KUKA KRL program: ho_st600_r1_1_2.src, ho_st600_r1_1_2.dat

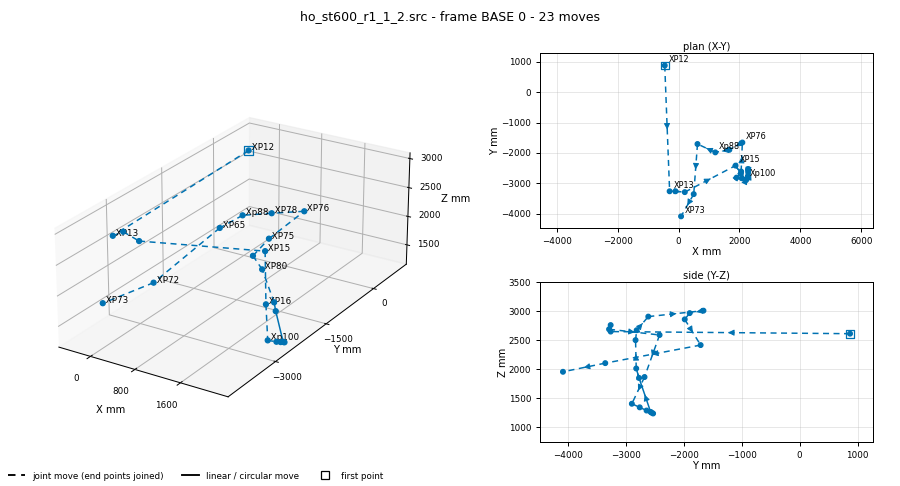
[picture p0: tool path of ho_st600_r1_1_2.src in frame BASE 0, 23 of 23 moves have a stored position in this frame; points joined in program order, loops and branches not executed]
--- ho_st600_r1_1_2.src ---
&ACCESS RVO1
&REL 137
&COMMENT Pega traseira ACTROS
&PARAM DISKPATH = KRC:\R1\Program\MANIPULACAO LTC
DEF ho_st600_r1_1_2( )
;FOLD INI
  ;FOLD BASISTECH INI
    GLOBAL INTERRUPT DECL 3 WHEN $STOPMESS==TRUE DO IR_STOPM ( )
    INTERRUPT ON 3
    BAS (#INITMOV,0 )
  ;ENDFOLD (BASISTECH INI)
;FOLD GRIPPERTECH INI
USER_GRP(0,DUMMY,DUMMY,GDEFAULT)
;ENDFOLD (GRIPPERTECH INI)
  ;FOLD USER INI
    ;Make your modifications here

  ;ENDFOLD (USER INI)
;ENDFOLD (INI)

; Caracterização dos meios de produção:
; Changes: Pega Traseira Actros
; Modelos: MGS\MGSB\LTA\LTB\STB
; Versão Atual: 22/07/2015
; Name: P13.050-R1

chk_w5_wechs_ok ( )              ; CHECK GRIPPER ACTROS

;FOLD PTP P12 CONT Vel=100 % PDAT11 Tool[5]:Painel Traseiro Actros Base[0];%{PE}%R 8.2.19,%MKUKATPBASIS,%CMOVE,%VPTP,%P 1:PTP, 2:P12, 3:C_DIS, 5:100, 7:PDAT11
$BWDSTART=FALSE
PDAT_ACT=PPDAT11
FDAT_ACT=FP12
BAS(#PTP_PARAMS,100)
PTP XP12 C_DIS
;ENDFOLD
;FOLD PTP P13 Vel=100 % PDAT12 Tool[5]:Painel Traseiro Actros Base[0];%{PE}%R 8.2.20,%MKUKATPBASIS,%CMOVE,%VPTP,%P 1:PTP, 2:P13, 3:, 5:100, 7:PDAT12
$BWDSTART=FALSE
PDAT_ACT=PPDAT12
FDAT_ACT=FP13
BAS(#PTP_PARAMS,100)
PTP XP13
;ENDFOLD

;FOLD OUT 3352 'R1 busca traseira' State=TRUE ;%{PE}%R 8.2.20,%MKUKATPBASIS,%COUT,%VOUTX,%P 2:3352, 3:R1 busca traseira, 5:TRUE, 6:
$OUT[3352]=TRUE
;ENDFOLD
;FOLD WAIT FOR ( IN 3352 'Aguarda lib. Buscar traseira' );%{PE}%R 8.2.20,%MKUKATPBASIS,%CEXT_WAIT_FOR,%VEXT_WAIT_FOR,%P 2:, 4:, 5:$IN, 6:3352, 7:Aguarda lib. Buscar traseira, 9:
WAIT FOR  ( $IN[3352] )
;ENDFOLD
;FOLD OUT 3352 'R1 busca traseira' State=FALSE ;%{PE}%R 8.2.20,%MKUKATPBASIS,%COUT,%VOUTX,%P 2:3352, 3:R1 busca traseira, 5:FALSE, 6:
$OUT[3352]=FALSE
;ENDFOLD

;FOLD PTP P74 Vel=100 % PDAT78 Tool[5]:Painel Traseiro Actros Base[0];%{PE}%R 8.2.20,%MKUKATPBASIS,%CMOVE,%VPTP,%P 1:PTP, 2:P74, 3:, 5:100, 7:PDAT78
$BWDSTART=FALSE
PDAT_ACT=PPDAT78
FDAT_ACT=FP74
BAS(#PTP_PARAMS,100)
PTP XP74
;ENDFOLD
;FOLD PTP P14 CONT Vel=100 % PDAT13 Tool[5]:Painel Traseiro Actros Base[0];%{PE}%R 8.2.19,%MKUKATPBASIS,%CMOVE,%VPTP,%P 1:PTP, 2:P14, 3:C_DIS, 5:100, 7:PDAT13
$BWDSTART=FALSE
PDAT_ACT=PPDAT13
FDAT_ACT=FP14
BAS(#PTP_PARAMS,100)
PTP XP14 C_DIS
;ENDFOLD
;FOLD PTP P15 CONT Vel=100 % PDAT14 Tool[5]:Painel Traseiro Actros Base[0];%{PE}%R 8.2.19,%MKUKATPBASIS,%CMOVE,%VPTP,%P 1:PTP, 2:P15, 3:C_DIS, 5:100, 7:PDAT14
$BWDSTART=FALSE
PDAT_ACT=PPDAT14
FDAT_ACT=FP15
BAS(#PTP_PARAMS,100)
PTP XP15 C_DIS
;ENDFOLD
;FOLD PTP P16 CONT Vel=100 % PDAT15 Tool[5]:Painel Traseiro Actros Base[0];%{PE}%R 8.2.19,%MKUKATPBASIS,%CMOVE,%VPTP,%P 1:PTP, 2:P16, 3:C_DIS, 5:100, 7:PDAT15
$BWDSTART=FALSE
PDAT_ACT=PPDAT15
FDAT_ACT=FP16
BAS(#PTP_PARAMS,100)
PTP XP16 C_DIS
;ENDFOLD

;FOLD OUT 3342 'Fora area externa' State=FALSE ;%{PE}%R 8.2.20,%MKUKATPBASIS,%COUT,%VOUTX,%P 2:3342, 3:Fora area externa, 5:FALSE, 6:
$OUT[3342]=FALSE
;ENDFOLD

;FOLD SET Z2.1/2 GRP ACTROS State= GDAT2;%{PE}%R 8.2.1,%MKUKATPGRP,%CGRP,%VGRP,%P 2:1, 4:1, 5:#NO, 6:GDAT2, 8:0, 10:0
H50(GRP,1,1,GGDAT2)
;ENDFOLD
chk_w5_grp2_opn()
;FOLD SET Z3.1/2 GRP ACTROS State=OPN GDAT3;%{PE}%R 8.2.1,%MKUKATPGRP,%CGRP,%VGRP,%P 2:2, 4:1, 5:#NO, 6:GDAT3, 8:0, 10:0
H50(GRP,2,1,GGDAT3)
;ENDFOLD
chk_w5_grp3_opn()

;FOLD PTP p100 CONT Vel=100 % PDAT71 Tool[5]:Painel Traseiro Actros Base[0];%{PE}%R 8.2.20,%MKUKATPBASIS,%CMOVE,%VPTP,%P 1:PTP, 2:p100, 3:C_DIS, 5:100, 7:PDAT71
$BWDSTART=FALSE
PDAT_ACT=PPDAT71
FDAT_ACT=Fp100
BAS(#PTP_PARAMS,100)
PTP Xp100 C_DIS
;ENDFOLD
;FOLD PTP p102 CONT Vel=100 % PDAT73 Tool[5]:Painel Traseiro Actros Base[0];%{PE}%R 8.2.20,%MKUKATPBASIS,%CMOVE,%VPTP,%P 1:PTP, 2:p102, 3:C_DIS, 5:100, 7:PDAT73
$BWDSTART=FALSE
PDAT_ACT=PPDAT73
FDAT_ACT=Fp102
BAS(#PTP_PARAMS,100)
PTP Xp102 C_DIS
;ENDFOLD
;FOLD PTP P82 Vel=100 % PDAT84 Tool[5]:Painel Traseiro Actros Base[0];%{PE}%R 8.2.20,%MKUKATPBASIS,%CMOVE,%VPTP,%P 1:PTP, 2:P82, 3:, 5:100, 7:PDAT84
$BWDSTART=FALSE
PDAT_ACT=PPDAT84
FDAT_ACT=FP82
BAS(#PTP_PARAMS,100)
PTP XP82
;ENDFOLD

;FOLD ; POSICAO DE PEGA DA PECA;%{PE}%R 8.2.20,%MKUKATPBASIS,%CCOMMENT,%VNORMAL,%P 2:POSICAO  DE  PEGA  DA  PECA
;ENDFOLD
;FOLD LIN P18 Vel=0.5 m/s CPDAT1 Tool[5]:Painel Traseiro Actros Base[0];%{PE}%R 8.2.20,%MKUKATPBASIS,%CMOVE,%VLIN,%P 1:LIN, 2:P18, 3:, 5:0.5, 7:CPDAT1
$BWDSTART=FALSE
LDAT_ACT=LCPDAT1
FDAT_ACT=FP18
BAS(#CP_PARAMS,0.5)
LIN XP18
;ENDFOLD

IF (NOT(GHOST())) THEN
;FOLD WAIT FOR ( IN 1 'Presença de peça 1 - Actros Todos' ) AND ( IN 2 'Presença de peça 2 - Actros Todos' );%{PE}%R 8.2.20,%MKUKATPBASIS,%CEXT_WAIT_FOR,%VEXT_WAIT_FOR,%P 2:, 4:, 5:$IN, 6:1, 7:Presença de peça 1 - Actros Todos, 9:AND, 10:, 12:, 13:$IN, 14:2, 15:Presença de peça 2 - Actros Todos, 17:
WAIT FOR  ( $IN[1] ) AND ( $IN[2] )
;ENDFOLD
ENDIF

;FOLD SET Z2.1/2 GRP ACTROS State=CLO GDAT1;%{PE}%R 8.2.1,%MKUKATPGRP,%CGRP,%VGRP,%P 2:1, 4:2, 5:#NO, 6:GDAT1, 8:0, 10:0
H50(GRP,1,2,GGDAT1)
;ENDFOLD
chk_w5_grp2_clo()
;FOLD SET Z3.1/2 GRP ACTROS State=CLO GDAT4;%{PE}%R 8.2.1,%MKUKATPGRP,%CGRP,%VGRP,%P 2:2, 4:2, 5:#NO, 6:GDAT4, 8:0, 10:0
H50(GRP,2,2,GGDAT4)
;ENDFOLD
chk_w5_grp3_clo()

IF (NOT(GHOST())) THEN
;FOLD SET Ventosa ACTROS State=VACUUM GDAT5;%{PE}%R 8.2.1,%MKUKATPGRP,%CGRP,%VGRP,%P 2:6, 4:1, 5:#NO, 6:GDAT5, 8:0, 10:0
H50(GRP,6,1,GGDAT5)
;ENDFOLD
;chk_w5_grp1_vac()
ENDIF

;FOLD OUT 3349 'R1 pegou peça' State=TRUE ;%{PE}%R 8.2.20,%MKUKATPBASIS,%COUT,%VOUTX,%P 2:3349, 3:R1 pegou peça, 5:TRUE, 6:
$OUT[3349]=TRUE
;ENDFOLD
;FOLD OUT 3350 'Solicita lib. sair magazine' State=TRUE ;%{PE}%R 8.2.20,%MKUKATPBASIS,%COUT,%VOUTX,%P 2:3350, 3:Solicita lib. sair magazine, 5:TRUE, 6:
$OUT[3350]=TRUE
;ENDFOLD
;FOLD WAIT FOR ( IN 3349 'Aguarda lib sair magazine' );%{PE}%R 8.2.20,%MKUKATPBASIS,%CEXT_WAIT_FOR,%VEXT_WAIT_FOR,%P 2:, 4:, 5:$IN, 6:3349, 7:Aguarda lib sair magazine, 9:
WAIT FOR  ( $IN[3349] )
;ENDFOLD
;FOLD OUT 3350 'Solicita lib sair magazine' State=FALSE ;%{PE}%R 8.2.20,%MKUKATPBASIS,%COUT,%VOUTX,%P 2:3350, 3:Solicita lib sair magazine, 5:FALSE, 6:
$OUT[3350]=FALSE
;ENDFOLD

;FOLD LIN P81 CONT Vel=1 m/s CPDAT16 Tool[5]:Painel Traseiro Actros Base[0];%{PE}%R 8.2.20,%MKUKATPBASIS,%CMOVE,%VLIN,%P 1:LIN, 2:P81, 3:C_DIS C_DIS, 5:1, 7:CPDAT16
$BWDSTART=FALSE
LDAT_ACT=LCPDAT16
FDAT_ACT=FP81
BAS(#CP_PARAMS,1)
LIN XP81 C_DIS C_DIS
;ENDFOLD
;FOLD LIN p101 CONT Vel=1 m/s CPDAT12 Tool[5]:Painel Traseiro Actros Base[0];%{PE}%R 8.2.20,%MKUKATPBASIS,%CMOVE,%VLIN,%P 1:LIN, 2:p101, 3:C_DIS C_DIS, 5:1, 7:CPDAT12
$BWDSTART=FALSE
LDAT_ACT=LCPDAT12
FDAT_ACT=Fp101
BAS(#CP_PARAMS,1)
LIN Xp101 C_DIS C_DIS
;ENDFOLD
;FOLD LIN P79 CONT Vel=2 m/s CPDAT15 Tool[5]:Painel Traseiro Actros Base[0];%{PE}%R 8.2.20,%MKUKATPBASIS,%CMOVE,%VLIN,%P 1:LIN, 2:P79, 3:C_DIS C_DIS, 5:2, 7:CPDAT15
$BWDSTART=FALSE
LDAT_ACT=LCPDAT15
FDAT_ACT=FP79
BAS(#CP_PARAMS,2)
LIN XP79 C_DIS C_DIS
;ENDFOLD
;FOLD LIN p95 CONT Vel=1 m/s CPDAT11 Tool[5]:Painel Traseiro Actros Base[0];%{PE}%R 8.2.20,%MKUKATPBASIS,%CMOVE,%VLIN,%P 1:LIN, 2:p95, 3:C_DIS C_DIS, 5:1, 7:CPDAT11
$BWDSTART=FALSE
LDAT_ACT=LCPDAT11
FDAT_ACT=Fp95
BAS(#CP_PARAMS,1)
LIN Xp95 C_DIS C_DIS
;ENDFOLD

IF (NOT(GHOST())) THEN
;FOLD WAIT FOR ( IN 1 'Presença de peça 1 - Actros Todos' ) AND ( IN 2 'Presença de peça 2 - Actros Todos' );%{PE}%R 8.2.20,%MKUKATPBASIS,%CEXT_WAIT_FOR,%VEXT_WAIT_FOR,%P 2:, 4:, 5:$IN, 6:1, 7:Presença de peça 1 - Actros Todos, 9:AND, 10:, 12:, 13:$IN, 14:2, 15:Presença de peça 2 - Actros Todos, 17:
WAIT FOR  ( $IN[1] ) AND ( $IN[2] )
;ENDFOLD
ENDIF

;FOLD PTP P80 CONT Vel=100 % PDAT83 Tool[5]:Painel Traseiro Actros Base[0];%{PE}%R 8.2.20,%MKUKATPBASIS,%CMOVE,%VPTP,%P 1:PTP, 2:P80, 3:C_DIS, 5:100, 7:PDAT83
$BWDSTART=FALSE
PDAT_ACT=PPDAT83
FDAT_ACT=FP80
BAS(#PTP_PARAMS,100)
PTP XP80 C_DIS
;ENDFOLD
;FOLD PTP P21 CONT Vel=100 % PDAT19 Tool[5]:Painel Traseiro Actros Base[0];%{PE}%R 8.2.19,%MKUKATPBASIS,%CMOVE,%VPTP,%P 1:PTP, 2:P21, 3:C_DIS, 5:100, 7:PDAT19
$BWDSTART=FALSE
PDAT_ACT=PPDAT19
FDAT_ACT=FP21
BAS(#PTP_PARAMS,100)
PTP XP21 C_DIS
;ENDFOLD
;FOLD PTP P75 CONT Vel=100 % PDAT79 Tool[5]:Painel Traseiro Actros Base[0];%{PE}%R 8.2.20,%MKUKATPBASIS,%CMOVE,%VPTP,%P 1:PTP, 2:P75, 3:C_DIS, 5:100, 7:PDAT79
$BWDSTART=FALSE
PDAT_ACT=PPDAT79
FDAT_ACT=FP75
BAS(#PTP_PARAMS,100)
PTP XP75 C_DIS
;ENDFOLD
;FOLD PTP P76 CONT Vel=100 % PDAT80 Tool[5]:Painel Traseiro Actros Base[0];%{PE}%R 8.2.20,%MKUKATPBASIS,%CMOVE,%VPTP,%P 1:PTP, 2:P76, 3:C_DIS, 5:100, 7:PDAT80
$BWDSTART=FALSE
PDAT_ACT=PPDAT80
FDAT_ACT=FP76
BAS(#PTP_PARAMS,100)
PTP XP76 C_DIS
;ENDFOLD
;FOLD PTP P78 CONT Vel=100 % PDAT82 Tool[5]:Painel Traseiro Actros Base[0];%{PE}%R 8.2.20,%MKUKATPBASIS,%CMOVE,%VPTP,%P 1:PTP, 2:P78, 3:C_DIS, 5:100, 7:PDAT82
$BWDSTART=FALSE
PDAT_ACT=PPDAT82
FDAT_ACT=FP78
BAS(#PTP_PARAMS,100)
PTP XP78 C_DIS
;ENDFOLD
;FOLD PTP p88 CONT Vel=100 % PDAT60 Tool[5]:Painel Traseiro Actros Base[0];%{PE}%R 8.2.19,%MKUKATPBASIS,%CMOVE,%VPTP,%P 1:PTP, 2:p88, 3:C_DIS, 5:100, 7:PDAT60
$BWDSTART=FALSE
PDAT_ACT=PPDAT60
FDAT_ACT=Fp88
BAS(#PTP_PARAMS,100)
PTP Xp88 C_DIS
;ENDFOLD
;FOLD PTP P65 CONT Vel=100 % PDAT74 Tool[5]:Painel Traseiro Actros Base[0];%{PE}%R 8.2.20,%MKUKATPBASIS,%CMOVE,%VPTP,%P 1:PTP, 2:P65, 3:C_DIS, 5:100, 7:PDAT74
$BWDSTART=FALSE
PDAT_ACT=PPDAT74
FDAT_ACT=FP65
BAS(#PTP_PARAMS,100)
PTP XP65 C_DIS
;ENDFOLD
;FOLD PTP P72 CONT Vel=100 % PDAT76 Tool[5]:Painel Traseiro Actros Base[0];%{PE}%R 8.2.20,%MKUKATPBASIS,%CMOVE,%VPTP,%P 1:PTP, 2:P72, 3:C_DIS, 5:100, 7:PDAT76
$BWDSTART=FALSE
PDAT_ACT=PPDAT76
FDAT_ACT=FP72
BAS(#PTP_PARAMS,100)
PTP XP72 C_DIS
;ENDFOLD

;FOLD Collision.Monitoring_AREA_5_On ;%{PE}%MKUKATPUSER
COLLSTOP( 11, 1 ) ;not Interrupt-Controlled
;ENDFOLD

;FOLD OUT 3349 'R1 Pegou peca' State=TRUE ;%{PE}%R 8.2.20,%MKUKATPBASIS,%COUT,%VOUTX,%P 2:3349, 3:R1 Pegou peca, 5:TRUE, 6:
$OUT[3349]=TRUE
;ENDFOLD
;FOLD OUT 3342 'Fora area externa' State=TRUE ;%{PE}%R 8.2.20,%MKUKATPBASIS,%COUT,%VOUTX,%P 2:3342, 3:Fora area externa, 5:TRUE, 6:
$OUT[3342]=TRUE
;ENDFOLD

;FOLD PTP P73 Vel=100 % PDAT77 Tool[5]:Painel Traseiro Actros Base[0];%{PE}%R 8.2.20,%MKUKATPBASIS,%CMOVE,%VPTP,%P 1:PTP, 2:P73, 3:, 5:100, 7:PDAT77
$BWDSTART=FALSE
PDAT_ACT=PPDAT77
FDAT_ACT=FP73
BAS(#PTP_PARAMS,100)
PTP XP73
;ENDFOLD

END

--- ho_st600_r1_1_2.dat ---
&ACCESS RVO1
&REL 137
&COMMENT Pega traseira ACTROS
&PARAM DISKPATH = KRC:\R1\Program\MANIPULACAO LTC
DEFDAT  ho_st600_r1_1_2
;FOLD EXTERNAL DECLARATIONS;%{PE}%MKUKATPBASIS,%CEXT,%VCOMMON,%P
;FOLD GRIPPERTECH EXT
EXT  H50 (INT  :IN,INT  :IN,INT  :IN,GRP_TYP  :IN )
;ENDFOLD (GRIPPERTECH EXT)
;FOLD SPOTTECH EXT
EXT  USERSPOT (S_COMMAND  :IN,SPOT_TYPE  :IN )
;ENDFOLD (SPOTTECH EXT)
;FOLD BASISTECH EXT;%{PE}%MKUKATPBASIS,%CEXT,%VEXT,%P
EXT  BAS (BAS_COMMAND  :IN,REAL  :IN )
DECL INT SUCCESS
;ENDFOLD (BASISTECH EXT)
;FOLD USER EXT;%{E}%MKUKATPUSER,%CEXT,%VEXT,%P
;Make your modifications here

;ENDFOLD (USER EXT)
;ENDFOLD (EXTERNAL DECLARATIONS)

;# ============ START PATH : bh_p13050r1_lta_01 =============
DECL BASIS_SUGG_T LAST_BASIS={POINT1[] "P82                     ",POINT2[] "P82                     ",CP_PARAMS[] "CPDAT0                  ",PTP_PARAMS[] "PDAT84                  ",CONT[] "                        ",CP_VEL[] "2.0                     ",PTP_VEL[] "100                     ",SYNC_PARAMS[] "SYNCDAT                 ",SPL_NAME[] "S0                      "}
DECL PDAT PPDAT11={VEL 100.0,ACC 100.0,APO_DIST 100.0,APO_MODE #CDIS}
DECL E6POS XP12={X -451.816589,Y 870.27887,Z 2616.43896,A -71.9595718,B 86.8192902,C 144.022598,S 2,T 11,E1 -267.097687,E2 0.0,E3 0.0,E4 0.0,E5 0.0,E6 0.0}
DECL FDAT FP12={TOOL_NO 5,BASE_NO 0,IPO_FRAME #BASE,POINT2[] " ",TQ_STATE FALSE}
DECL PDAT PPDAT12={VEL 100.0,ACC 100.0,APO_DIST 100.0,APO_MODE #CDIS}
DECL E6POS XP13={X -291.739288,Y -3257.74512,Z 2653.0061,A 20.6638298,B 86.1274414,C -123.413696,S 2,T 11,E1 -4438.05518,E2 0.0,E3 0.0,E4 0.0,E5 0.0,E6 0.0}
DECL FDAT FP13={TOOL_NO 5,BASE_NO 0,IPO_FRAME #BASE,POINT2[] " ",TQ_STATE FALSE}
DECL PDAT PPDAT13={VEL 100.0,ACC 100.0,APO_DIST 100.0,APO_MODE #CDIS}
DECL E6POS XP14={X 205.846802,Y -3285.1731,Z 2693.19409,A -3.17952704,B 85.6848679,C -123.935898,S 2,T 11,E1 -4438.06104,E2 0.0,E3 0.0,E4 0.0,E5 0.0,E6 0.0}
DECL FDAT FP14={TOOL_NO 5,BASE_NO 0,IPO_FRAME #BASE,POINT2[] " ",TQ_STATE FALSE}
DECL PDAT PPDAT14={VEL 100.0,ACC 100.0,APO_DIST 100.0,APO_MODE #CDIS}
DECL E6POS XP15={X 1872.49097,Y -2414.4231,Z 2594.0769,A -19.4102993,B 84.5822067,C -109.933098,S 2,T 11,E1 -3412.81689,E2 0.0,E3 0.0,E4 0.0,E5 0.0,E6 0.0}
DECL FDAT FP15={TOOL_NO 5,BASE_NO 0,IPO_FRAME #BASE,POINT2[] " ",TQ_STATE FALSE}
DECL PDAT PPDAT15={VEL 100.0,ACC 100.0,APO_DIST 100.0,APO_MODE #CDIS}
DECL E6POS XP16={X 2049.04297,Y -2673.92407,Z 1868.73901,A -84.6288071,B 74.7002335,C -174.507401,S 2,T 11,E1 -3291.271,E2 0.0,E3 0.0,E4 0.0,E5 0.0,E6 0.0}
DECL FDAT FP16={TOOL_NO 5,BASE_NO 0,IPO_FRAME #BASE,POINT2[] " ",TQ_STATE FALSE}
DECL LDAT LCPDAT1={VEL 2.0,ACC 100.0,APO_DIST 100.0,APO_FAC 50.0,AXIS_VEL 100.0,AXIS_ACC 100.0,ORI_TYP #VAR,CIRC_TYP #BASE,JERK_FAC 50.0,GEAR_JERK 50.0,EXAX_IGN 0}
DECL E6POS XP18={X 2287.61304,Y -2526.11206,Z 1240.37695,A -89.8074493,B 66.0794296,C -179.626907,S 2,T 11,E1 -3241.46289,E2 0.0,E3 0.0,E4 0.0,E5 0.0,E6 0.0}
DECL FDAT FP18={TOOL_NO 5,BASE_NO 0,IPO_FRAME #BASE,POINT2[] " ",TQ_STATE FALSE}
DECL E6POS XP21={X 1903.797,Y -2809.604,Z 2675.91406,A -52.9545403,B 81.9597015,C -137.800507,S 2,T 11,E1 -3600.21191,E2 0.0,E3 0.0,E4 0.0,E5 0.0,E6 0.0}
DECL FDAT FP21={TOOL_NO 5,BASE_NO 0,IPO_FRAME #BASE,POINT2[] " ",TQ_STATE FALSE}
DECL PDAT PPDAT19={VEL 100.0,ACC 100.0,APO_DIST 100.0,APO_MODE #CDIS}
DECL E6POS XP88={X 1207.65796,Y -1980.32104,Z 2863.53809,A 30.6810093,B 83.3284302,C 30.6459599,S 2,T 10,E1 -964.773499,E2 0.0,E3 0.0,E4 0.0,E5 0.0,E6 0.0}
DECL FDAT Fp88={TOOL_NO 5,BASE_NO 0,IPO_FRAME #BASE,POINT2[] " ",TQ_STATE FALSE}
DECL PDAT PPDAT60={VEL 100.0,ACC 100.0,APO_DIST 100.0,APO_MODE #CDIS}
DECL E6POS XP95={X 2276.68311,Y -2816.91406,Z 2016.46301,A -88.0621414,B 73.5641479,C -177.631104,S 2,T 11,E1 -3601.14893,E2 0.0,E3 0.0,E4 0.0,E5 0.0,E6 0.0}
DECL FDAT Fp95={TOOL_NO 5,BASE_NO 0,IPO_FRAME #BASE,POINT2[] " ",TQ_STATE FALSE}
DECL LDAT LCPDAT11={VEL 2.0,ACC 100.0,APO_DIST 100.0,APO_FAC 50.0,AXIS_VEL 100.0,AXIS_ACC 100.0,ORI_TYP #VAR,CIRC_TYP #BASE,JERK_FAC 50.0,GEAR_JERK 50.0,EXAX_IGN 0}
DECL GRP_SUGG_T LAST_GRP={NUMBER[] "6                       ",STATE[] "1                       ",PARAMS[] "GDAT5                   "}
DECL GRP_TYP GGDAT1={G_APO #NO,GRP_TIME 0.200000003,CTRL #OFF,DLY 0,DST 1}
DECL GRP_TYP GGDAT2={G_APO #NO,GRP_TIME 0.200000003,CTRL #OFF,DLY 0,DST 1}
DECL GRP_TYP GGDAT3={G_APO #NO,GRP_TIME 0.200000003,CTRL #OFF,DLY 0,DST 1}
DECL GRP_TYP GGDAT4={G_APO #NO,GRP_TIME 0.200000003,CTRL #OFF,DLY 0,DST 1}
DECL PDAT PPDAT71={VEL 100.0,ACC 100.0,APO_DIST 100.0,APO_MODE #CDIS}
DECL E6POS Xp100={X 2215.93408,Y -2892.56909,Z 1408.06995,A -88.7884293,B 64.9466476,C -178.740005,S 2,T 11,E1 -3241.45508,E2 0.0,E3 0.0,E4 0.0,E5 0.0,E6 0.0}
DECL FDAT Fp100={TOOL_NO 5,BASE_NO 0,IPO_FRAME #BASE,POINT2[] " ",TQ_STATE FALSE}
DECL GRP_TYP GGDAT5={G_APO #NO,GRP_TIME 0.200000003,CTRL #OFF,DLY 0,DST 1}
DECL E6POS XP101={X 2288.98999,Y -2568.38989,Z 1266.61902,A -89.3097763,B 65.7357788,C -179.678497,S 2,T 11,E1 -3241.45703,E2 0.0,E3 0.0,E4 0.0,E5 0.0,E6 0.0}
DECL FDAT Fp101={TOOL_NO 5,BASE_NO 0,IPO_FRAME #BASE,POINT2[] " ",TQ_STATE FALSE}
DECL LDAT LCPDAT12={VEL 2.0,ACC 100.0,APO_DIST 100.0,APO_FAC 50.0,AXIS_VEL 100.0,AXIS_ACC 100.0,ORI_TYP #VAR,CIRC_TYP #BASE,JERK_FAC 50.0,GEAR_JERK 50.0,EXAX_IGN 0}
DECL E6POS XP102={X 2285.14893,Y -2756.62891,Z 1346.18201,A -89.3083572,B 65.7357483,C -179.677094,S 2,T 11,E1 -3241.45996,E2 0.0,E3 0.0,E4 0.0,E5 0.0,E6 0.0}
DECL FDAT Fp102={TOOL_NO 5,BASE_NO 0,IPO_FRAME #BASE,POINT2[] " ",TQ_STATE FALSE}
DECL PDAT PPDAT73={VEL 100.0,ACC 80.0,APO_DIST 50.0,APO_MODE #CDIS}
DECL E6POS XP65={X 622.74469,Y -1706.19104,Z 2420.0,A 49.025631,B 84.2697983,C 62.7197914,S 2,T 10,E1 -486.5271,E2 0.0,E3 0.0,E4 0.0,E5 0.0,E6 0.0}
DECL FDAT FP65={TOOL_NO 5,BASE_NO 0,IPO_FRAME #BASE,POINT2[] " ",TQ_STATE FALSE}
DECL PDAT PPDAT74={VEL 100.0,ACC 100.0,APO_DIST 20.0,APO_MODE #CDIS}
DECL E6POS XP72={X 499.292694,Y -3351.04712,Z 2108.56812,A -9.71163654,B 86.2505112,C 11.5372105,S 2,T 10,E1 -1946.46802,E2 0.0,E3 0.0,E4 0.0,E5 0.0,E6 0.0}
DECL FDAT FP72={TOOL_NO 5,BASE_NO 0,IPO_FRAME #BASE,POINT2[] " ",TQ_STATE FALSE}
DECL PDAT PPDAT76={VEL 100.0,ACC 50.0,APO_DIST 10.0,APO_MODE #CDIS}
DECL E6POS XP73={X 83.9855728,Y -4080.39502,Z 1959.36804,A 36.7836418,B 88.5122375,C 81.7560196,S 2,T 10,E1 -2701.97412,E2 0.0,E3 0.0,E4 0.0,E5 0.0,E6 0.0}
DECL FDAT FP73={TOOL_NO 5,BASE_NO 0,IPO_FRAME #BASE,POINT2[] " ",TQ_STATE FALSE}
DECL PDAT PPDAT77={VEL 100.0,ACC 100.0,APO_DIST 100.0,APO_MODE #CDIS}
DECL E6POS XP74={X -98.997879,Y -3257.86792,Z 2764.84399,A 36.1262589,B 77.7119293,C -97.4505692,S 2,T 11,E1 -4438.05713,E2 0.0,E3 0.0,E4 0.0,E5 0.0,E6 0.0}
DECL FDAT FP74={TOOL_NO 5,BASE_NO 0,IPO_FRAME #BASE,POINT2[] " ",TQ_STATE FALSE}
DECL PDAT PPDAT78={VEL 100.0,ACC 100.0,APO_DIST 100.0,APO_MODE #CDIS}
DECL E6POS XP75={X 2055.39893,Y -2608.81299,Z 2911.28296,A 46.0131302,B 78.8642807,C -23.3656807,S 2,T 11,E1 -3429.2019,E2 0.0,E3 0.0,E4 0.0,E5 0.0,E6 0.0}
DECL FDAT FP75={TOOL_NO 5,BASE_NO 0,IPO_FRAME #BASE,POINT2[] " ",TQ_STATE FALSE}
DECL PDAT PPDAT79={VEL 100.0,ACC 100.0,APO_DIST 100.0,APO_MODE #CDIS}
DECL E6POS XP76={X 2095.78003,Y -1657.45496,Z 3013.73193,A 64.6596985,B 73.4026337,C 0.0733646974,S 2,T 11,E1 -2471.62109,E2 0.0,E3 0.0,E4 0.0,E5 0.0,E6 0.0}
DECL FDAT FP76={TOOL_NO 5,BASE_NO 0,IPO_FRAME #BASE,POINT2[] " ",TQ_STATE FALSE}
DECL PDAT PPDAT80={VEL 100.0,ACC 100.0,APO_DIST 100.0,APO_MODE #CDIS}
DECL E6POS XP78={X 1668.724,Y -1895.37305,Z 2971.32788,A 17.5263195,B 78.23629,C 10.0105896,S 2,T 10,E1 -990.161987,E2 0.0,E3 0.0,E4 0.0,E5 0.0,E6 0.0}
DECL FDAT FP78={TOOL_NO 5,BASE_NO 0,IPO_FRAME #BASE,POINT2[] " ",TQ_STATE FALSE}
DECL PDAT PPDAT82={VEL 100.0,ACC 100.0,APO_DIST 100.0,APO_MODE #CDIS}
DECL E6POS XP79={X 2276.21899,Y -2768.38403,Z 1852.85999,A -88.4287796,B 71.8257599,C -178.175705,S 2,T 11,E1 -3521.24805,E2 0.0,E3 0.0,E4 0.0,E5 0.0,E6 0.0}
DECL FDAT FP79={TOOL_NO 5,BASE_NO 0,IPO_FRAME #BASE,POINT2[] " ",TQ_STATE FALSE}
DECL LDAT LCPDAT15={VEL 2.0,ACC 100.0,APO_DIST 100.0,APO_FAC 50.0,AXIS_VEL 100.0,AXIS_ACC 100.0,ORI_TYP #VAR,CIRC_TYP #BASE,JERK_FAC 50.0,GEAR_JERK 50.0,EXAX_IGN 0}
DECL E6POS XP80={X 2074.96509,Y -2828.56201,Z 2505.68506,A -68.1553726,B 80.0709534,C -153.210495,S 2,T 11,E1 -3600.46509,E2 0.0,E3 0.0,E4 0.0,E5 0.0,E6 0.0}
DECL FDAT FP80={TOOL_NO 5,BASE_NO 0,IPO_FRAME #BASE,POINT2[] " ",TQ_STATE FALSE}
DECL PDAT PPDAT83={VEL 100.0,ACC 100.0,APO_DIST 100.0,APO_MODE #CDIS}
DECL E6POS XP81={X 2287.50708,Y -2553.34692,Z 1255.51196,A -89.7614212,B 65.7057266,C -179.906204,S 2,T 11,E1 -3241.46606,E2 0.0,E3 0.0,E4 0.0,E5 0.0,E6 0.0}
DECL FDAT FP81={TOOL_NO 5,BASE_NO 0,IPO_FRAME #BASE,POINT2[] " ",TQ_STATE FALSE}
DECL LDAT LCPDAT16={VEL 2.0,ACC 100.0,APO_DIST 100.0,APO_FAC 50.0,AXIS_VEL 100.0,AXIS_ACC 100.0,ORI_TYP #VAR,CIRC_TYP #BASE,JERK_FAC 50.0,GEAR_JERK 50.0,EXAX_IGN 0}
DECL E6POS XP82={X 2287.18799,Y -2638.47192,Z 1291.22803,A -89.8141098,B 65.649437,C -179.632996,S 2,T 11,E1 -3241.46411,E2 0.0,E3 0.0,E4 0.0,E5 0.0,E6 0.0}
DECL FDAT FP82={TOOL_NO 5,BASE_NO 0,IPO_FRAME #BASE,POINT2[] " ",TQ_STATE FALSE}
DECL PDAT PPDAT84={VEL 100.0,ACC 100.0,APO_DIST 100.0,APO_MODE #CDIS}
ENDDAT
